TYPE StepCondition :
STRUCT
	name			: STRING;
	condition		: Condition;
//	nextAction		: STRING;
//	timeout			: TIME;
//	timeoutAction	: STRING;
	/// these will go to binding
END_STRUCT
END_TYPE

(* stored: Version 1.1.0.1, ProductVersion 3.1.4024.11
   DUT StepCondition: Id {e3fc571e-3dd2-4adb-87b0-7d7cbf833633} *)
